PROGRAM MAIN
VAR
	bPiezaOK: BOOL := FALSE;
	iContadorPiezaOK: INT;
END_VAR

IF bPiezaOK THEN
	iContadorPiezaOK := iContadorPiezaOK + 1;
END_IF

END_PROGRAM

(* stored: Version 1.1.0.1, ProductVersion 3.1.4024.16
   POU MAIN: Id {e9026f2b-3203-4a90-ba7a-cbef7540c309}, SpecialFunc None *)
